(* LS Electric XG5000 project: PLC *)
(* PLC LSPLC *)

PROGRAM NewProgram (* task: 스캔 프로그램 *)
VAR
    Array_g : ARRAY[0..9] OF INT;
    Array_w : ARRAY[0..9] OF INT;
    FIFO_g : FIFO_INT;
    FIFO_w : FIFO_INT;
    grade AT %MW800 : INT;
    INST : TOF;
    INST1 : TOF;
    INST10 : TOF;
    INST11 : TOF;
    INST12 : TOF;
    INST13 : TOF;
    INST14 : TOF;
    INST15 : TOF;
    INST16 : TOF;
    INST17 : TOF;
    INST18 : TOF;
    INST19 : TOF;
    INST2 : TOF;
    INST20 : TOF;
    INST21 : TON;
    INST22 : TON;
    INST23 : TON;
    INST24 : TOF;
    INST25 : TON;
    INST26 : TON;
    INST27 : TON;
    INST28 : TON;
    INST29 : TON;
    INST3 : TOF;
    INST30 : TON;
    INST31 : TON;
    INST32 : TON;
    INST33 : TON;
    INST34 : TON;
    INST35 : TON;
    INST36 : TON;
    INST37 : TON;
    INST38 : TON;
    INST39 : TON;
    INST4 : TOF;
    INST40 : TON;
    INST41 : TON;
    INST42 : TON;
    INST43 : TON;
    INST44 : TON;
    INST45 : TON;
    INST46 : TON;
    INST47 : TON;
    INST48 : TON;
    INST49 : TON;
    INST5 : TOF;
    INST50 : TON;
    INST51 : TON;
    INST52 : TON;
    INST53 : TON;
    INST54 : TON;
    INST55 : TON;
    INST56 : TON;
    INST6 : TOF;
    INST7 : TOF;
    INST8 : TOF;
    INST9 : TOF;
    INT1_g : INT;
    INT1_w : INT;
    INT2_g : INT;
    INT2_w : INT;
    INT_w : INT;
    IN_ARY AT %MW0 : ARRAY[0..3] OF INT;
    R : BOOL;
    STOP AT %IX0.0.1 : BOOL;
    STR1 : STRING;
    STR2 : STRING;
    SYSTEM_ON AT %IX0.0.0 : BOOL;
    weight AT %MW700 : INT;
    고_1_signal : BOOL;
    고_1_적재 : TON;
    고_1_적재량 : CTU_INT;
    고_1_적재상황 AT %QW0.3.0 : INT;
    고_2_signal : BOOL;
    고_2_적재 : TON;
    고_2_적재량 : CTU_INT;
    고_2_적재상황 AT %QW0.3.1 : INT;
    고_3_signal : BOOL;
    고_3_적재량 : CTU_INT;
    고_3_적재상황 AT %QW0.3.2 : INT;
    등급난수생성 : TON;
    등급난수생성1 : TON;
    라인 AT %QX0.1.30 : BOOL;
    무게난수생성 : TON;
    무게난수생성1 : TON;
    바닥1 AT %MX13 : BOOL;
    바닥1_a AT %QW0.6.3 : INT;
    바닥1_작동 : TON;
    바닥2 AT %MX14 : BOOL;
    바닥2_a AT %QW0.7.0 : INT;
    바닥2_작동 : TON;
    바닥3 AT %MX15 : BOOL;
    바닥3_a AT %QW0.7.1 : INT;
    바닥3_작동 : TON;
    바닥4 AT %MX16 : BOOL;
    바닥4_a AT %QW0.7.2 : INT;
    바닥4_작동 : TON;
    바닥5 AT %MX17 : BOOL;
    바닥5_a AT %QW0.7.3 : INT;
    바닥5_작동 : TON;
    바닥6 AT %MX18 : BOOL;
    바닥6_a AT %QW0.8.0 : INT;
    바닥6_작동 : TON;
    바닥7 AT %MX19 : BOOL;
    바닥7_a AT %QW0.8.1 : INT;
    바닥7_작동 : TON;
    바닥8 AT %MX20 : BOOL;
    바닥8_a AT %QW0.8.2 : INT;
    바닥8_작동 : TON;
    바닥9 AT %MX21 : BOOL;
    바닥9_a AT %QW0.8.3 : INT;
    바닥9_작동 : TON;
    바닥_9_적재 : TON;
    분류로봇1 AT %MX500 : BOOL;
    분류로봇1_작동 : TOF;
    분류로봇2 AT %MX510 : BOOL;
    분류로봇2_작동 : TOF;
    분류로봇3 AT %MX520 : BOOL;
    분류로봇3_작동 : TOF;
    분류로봇4 AT %MX530 : BOOL;
    분류로봇4_작동 : TOF;
    분류로봇5 AT %MX540 : BOOL;
    분류로봇5_작동 : TOF;
    분류로봇6 AT %MX550 : BOOL;
    분류로봇6_작동 : TOF;
    삼_고_적재상황 AT %QW1.3.2 : INT;
    삼_저_적재상황 AT %QW1.3.0 : INT;
    삼_중_적재상황 AT %QW1.3.1 : INT;
    생산_signal : BOOL;
    생산_signal_a AT %QW0.4.0 : INT;
    소터1 AT %MX4 : BOOL;
    소터10 AT %MX12 : BOOL;
    소터10_a AT %QW0.6.2 : INT;
    소터10_작동 : TON;
    소터11_작동 : TON;
    소터12_작동 : TON;
    소터13_작동 : TON;
    소터14_작동 : TON;
    소터1_a AT %QW0.4.1 : INT;
    소터1_작동 : TON;
    소터2 AT %MW20 : INT;
    소터2_a AT %QW0.4.2 : INT;
    소터2_신호 AT %QW0.9.0 : INT;
    소터3 AT %MX5 : BOOL;
    소터3_a AT %QW0.4.3 : INT;
    소터3_작동 : TON;
    소터4 AT %MX6 : BOOL;
    소터4_a AT %QW0.5.0 : INT;
    소터4_작동 : TON;
    소터5 AT %MX7 : BOOL;
    소터5_a AT %QW0.5.1 : INT;
    소터5_작동 : TON;
    소터6 AT %MX8 : BOOL;
    소터6_a AT %QW0.5.2 : INT;
    소터6_작동 : TON;
    소터7 AT %MX9 : BOOL;
    소터7_a AT %QW0.5.3 : INT;
    소터7_작동 : TON;
    소터8 AT %MX10 : BOOL;
    소터8_a AT %QW0.6.0 : INT;
    소터8_작동 : TON;
    소터9 AT %MX11 : BOOL;
    소터9_a AT %QW0.6.1 : INT;
    소터9_작동 : TON;
    신호 AT %MX400 : BOOL;
    신호1 : BOOL;
    이_고_적재상황 AT %QW1.2.2 : INT;
    이_저_적재상황 AT %QW1.2.0 : INT;
    이_중_적재상황 AT %QW1.2.1 : INT;
    일_고_적재상황 AT %QW1.1.2 : INT;
    일_저_적재상황 AT %QW1.1.0 : INT;
    일_중_적재상황 AT %QW1.1.1 : INT;
    재생산_delay : TOF;
    재생산_signal AT %MX350 : BOOL;
    저_1_signal : BOOL;
    저_1_적재 : TON;
    저_1_적재량 : CTU_INT;
    저_1_적재상황 AT %QW0.1.0 : INT;
    저_2_signal : BOOL;
    저_2_적재 : TON;
    저_2_적재량 : CTU_INT;
    저_2_적재상황 AT %QW0.1.1 : INT;
    저_3_signal : BOOL;
    저_3_적재 : TON;
    저_3_적재량 : CTU_INT;
    저_3_적재상황 AT %QW0.1.2 : INT;
    저_4_적재량 : CTU_INT;
    저_5_적재량 : CTU_INT;
    저_6_적재량 : CTU_INT;
    저_7_적재량 : CTU_INT;
    저_8_적재량 : CTU_INT;
    저_9_적재 : TON;
    저_9_적재량 : CTU_INT;
    제품생산 : TP;
    중_1_signal : BOOL;
    중_1_적재 : TON;
    중_1_적재량 : CTU_INT;
    중_1_적재상황 AT %QW0.2.0 : INT;
    중_2_signal : BOOL;
    중_2_적재 : TON;
    중_2_적재량 : CTU_INT;
    중_2_적재상황 AT %QW0.2.1 : INT;
    중_3_signal : BOOL;
    중_3_적재량 : CTU_INT;
    중_3_적재상황 AT %QW0.2.2 : INT;
    품질로봇 AT %MW30 : INT;
    품질로봇가동 : TOF;
    품질로봇대기 : TON;
END_VAR
VAR
    _t1 : BOOL;
    _e2 : R_TRIG;
    _e3 : F_TRIG;
    _e4 : R_TRIG;
    _e5 : F_TRIG;
    _e6 : F_TRIG;
    _e7 : R_TRIG;
    _t8 : BOOL;
    _t9 : BOOL;
    _t10 : BOOL;
    _t11 : BOOL;
    _t12 : DINT;
    _t13 : BOOL;
    _t14 : BOOL;
    _t15 : BOOL;
    _t16 : BOOL;
    _t17 : BOOL;
    _t18 : DINT;
    _t19 : BOOL;
    _t20 : BOOL;
    _t21 : BOOL;
    _t22 : BOOL;
    _t23 : BOOL;
    _t24 : DINT;
    _t25 : BOOL;
    _t26 : BOOL;
    _t27 : BOOL;
    _t28 : BOOL;
    _t29 : BOOL;
    _t30 : BOOL;
    _t31 : BOOL;
    _t32 : BOOL;
    _t33 : BOOL;
    _t34 : BOOL;
    _t35 : BOOL;
    _t36 : BOOL;
    _e37 : R_TRIG;
    _e38 : R_TRIG;
    _e39 : R_TRIG;
    _e40 : R_TRIG;
    _e41 : R_TRIG;
    _e42 : R_TRIG;
    _e43 : R_TRIG;
    _e44 : R_TRIG;
    _e45 : R_TRIG;
    _t46 : BOOL;
END_VAR

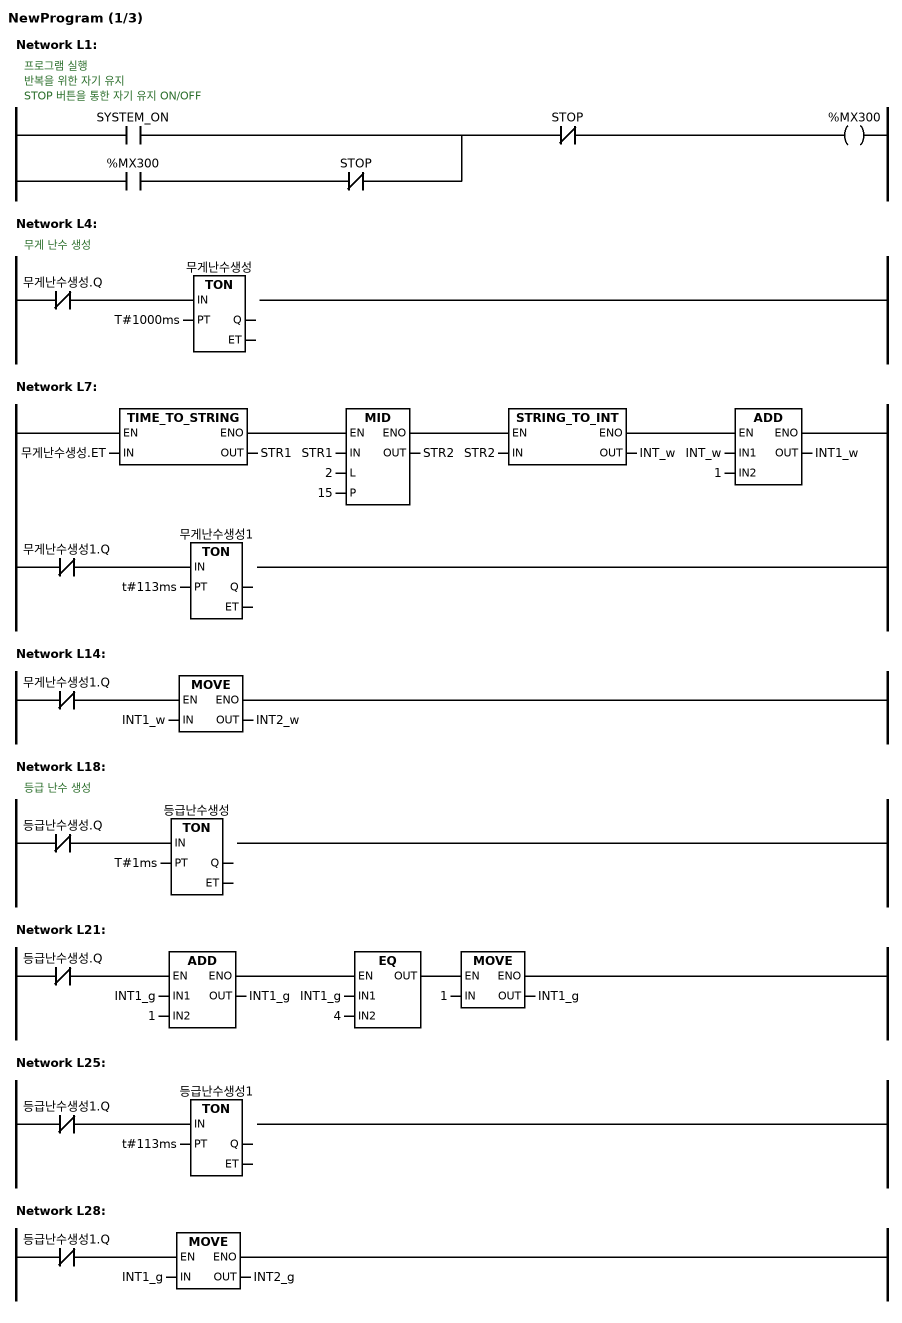
(* 프로그램 실행 / 반복을 위한 자기 유지 / STOP 버튼을 통한 자기 유지 ON/OFF *)
(* Rung L1 *)
%MX300 := (SYSTEM_ON OR (%MX300 AND NOT STOP)) AND NOT STOP;
(* 무게 난수 생성 *)
(* Rung L4 *)
무게난수생성(IN := NOT 무게난수생성.Q, PT := T#1000ms);
(* Rung L7 *)
STR1 := TIME_TO_STRING(무게난수생성.ET);
STR2 := MID(IN := STR1, L := 2, P := 15);
INT_w := STRING_TO_INT(STR2);
INT1_w := INT_w + 1;
무게난수생성1(IN := NOT 무게난수생성1.Q, PT := t#113ms);
(* Rung L14 *)
IF NOT 무게난수생성1.Q THEN INT2_w := INT1_w; END_IF;
(* 등급 난수 생성 *)
(* Rung L18 *)
등급난수생성(IN := NOT 등급난수생성.Q, PT := T#1ms);
(* Rung L21 *)
IF NOT 등급난수생성.Q THEN
    INT1_g := INT1_g + 1;
    _t1 := INT1_g = 4;
END_IF;
IF _t1 THEN INT1_g := 1; END_IF;
(* Rung L25 *)
등급난수생성1(IN := NOT 등급난수생성1.Q, PT := t#113ms);
(* Rung L28 *)
IF NOT 등급난수생성1.Q THEN INT2_g := INT1_g; END_IF;

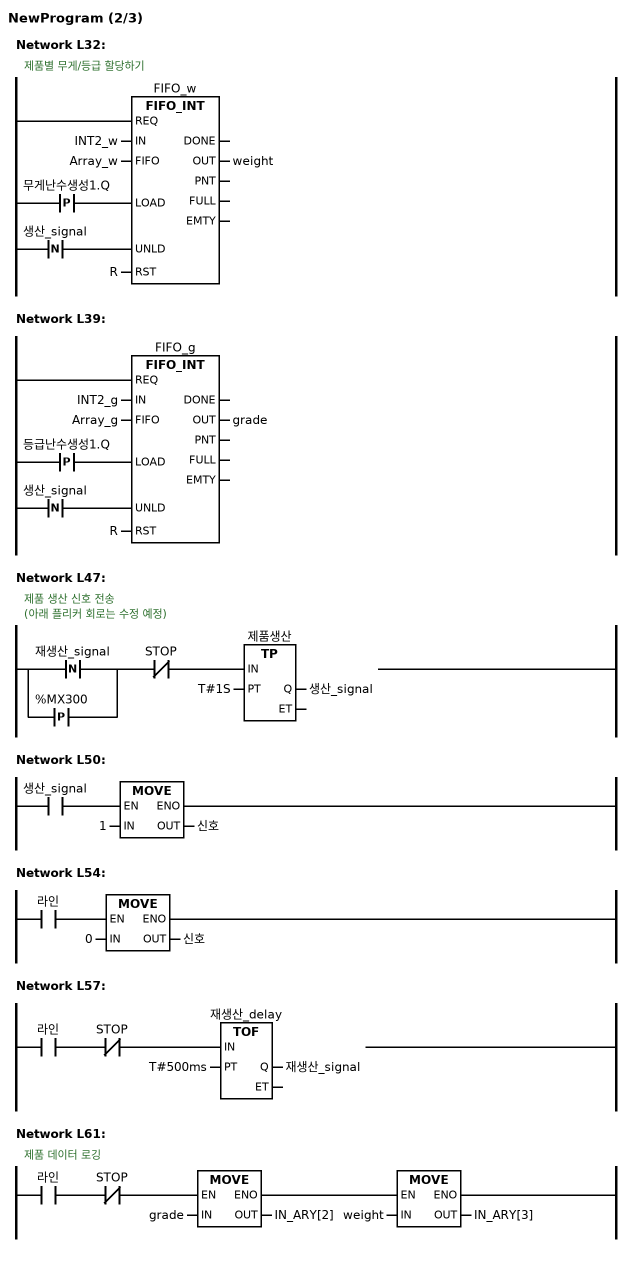
(* 제품별 무게/등급 할당하기 *)
(* Rung L32 *)
_e2(CLK := 무게난수생성1.Q);
_e3(CLK := 생산_signal);
FIFO_w(REQ := TRUE, IN := INT2_w, FIFO := Array_w, LOAD := _e2.Q, UNLD := _e3.Q, RST := R, OUT => weight);
(* Rung L39 *)
_e4(CLK := 등급난수생성1.Q);
_e5(CLK := 생산_signal);
FIFO_g(REQ := TRUE, IN := INT2_g, FIFO := Array_g, LOAD := _e4.Q, UNLD := _e5.Q, RST := R, OUT => grade);
(* 제품 생산 신호 전송 / (아래 플리커 회로는 수정 예정) *)
(* Rung L47 *)
_e6(CLK := 재생산_signal);
_e7(CLK := %MX300);
제품생산(IN := (_e6.Q OR _e7.Q) AND NOT STOP, PT := T#1S, Q => 생산_signal);
(* Rung L50 *)
IF 생산_signal THEN 신호 := 1; END_IF;
(* Rung L54 *)
IF 라인 THEN 신호 := 0; END_IF;
(* Rung L57 *)
재생산_delay(IN := 라인 AND NOT STOP, PT := T#500ms, Q => 재생산_signal);
(* 제품 데이터 로깅 *)
(* Rung L61 *)
IF 라인 AND NOT STOP THEN
    IN_ARY[2] := grade;
    IN_ARY[3] := weight;
END_IF;

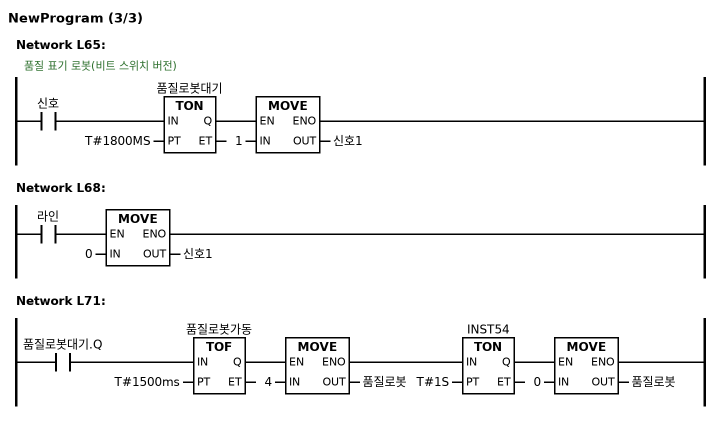
(* 품질 표기 로봇(비트 스위치 버전) *)
(* Rung L65 *)
품질로봇대기(IN := 신호, PT := T#1800MS);
IF 품질로봇대기.Q THEN 신호1 := 1; END_IF;
(* Rung L68 *)
IF 라인 THEN 신호1 := 0; END_IF;
(* Rung L71 *)
품질로봇가동(IN := 품질로봇대기.Q, PT := T#1500ms);
IF 품질로봇가동.Q THEN 품질로봇 := 4; END_IF;
INST54(IN := 품질로봇가동.Q, PT := T#1S);
IF INST54.Q THEN 품질로봇 := 0; END_IF;

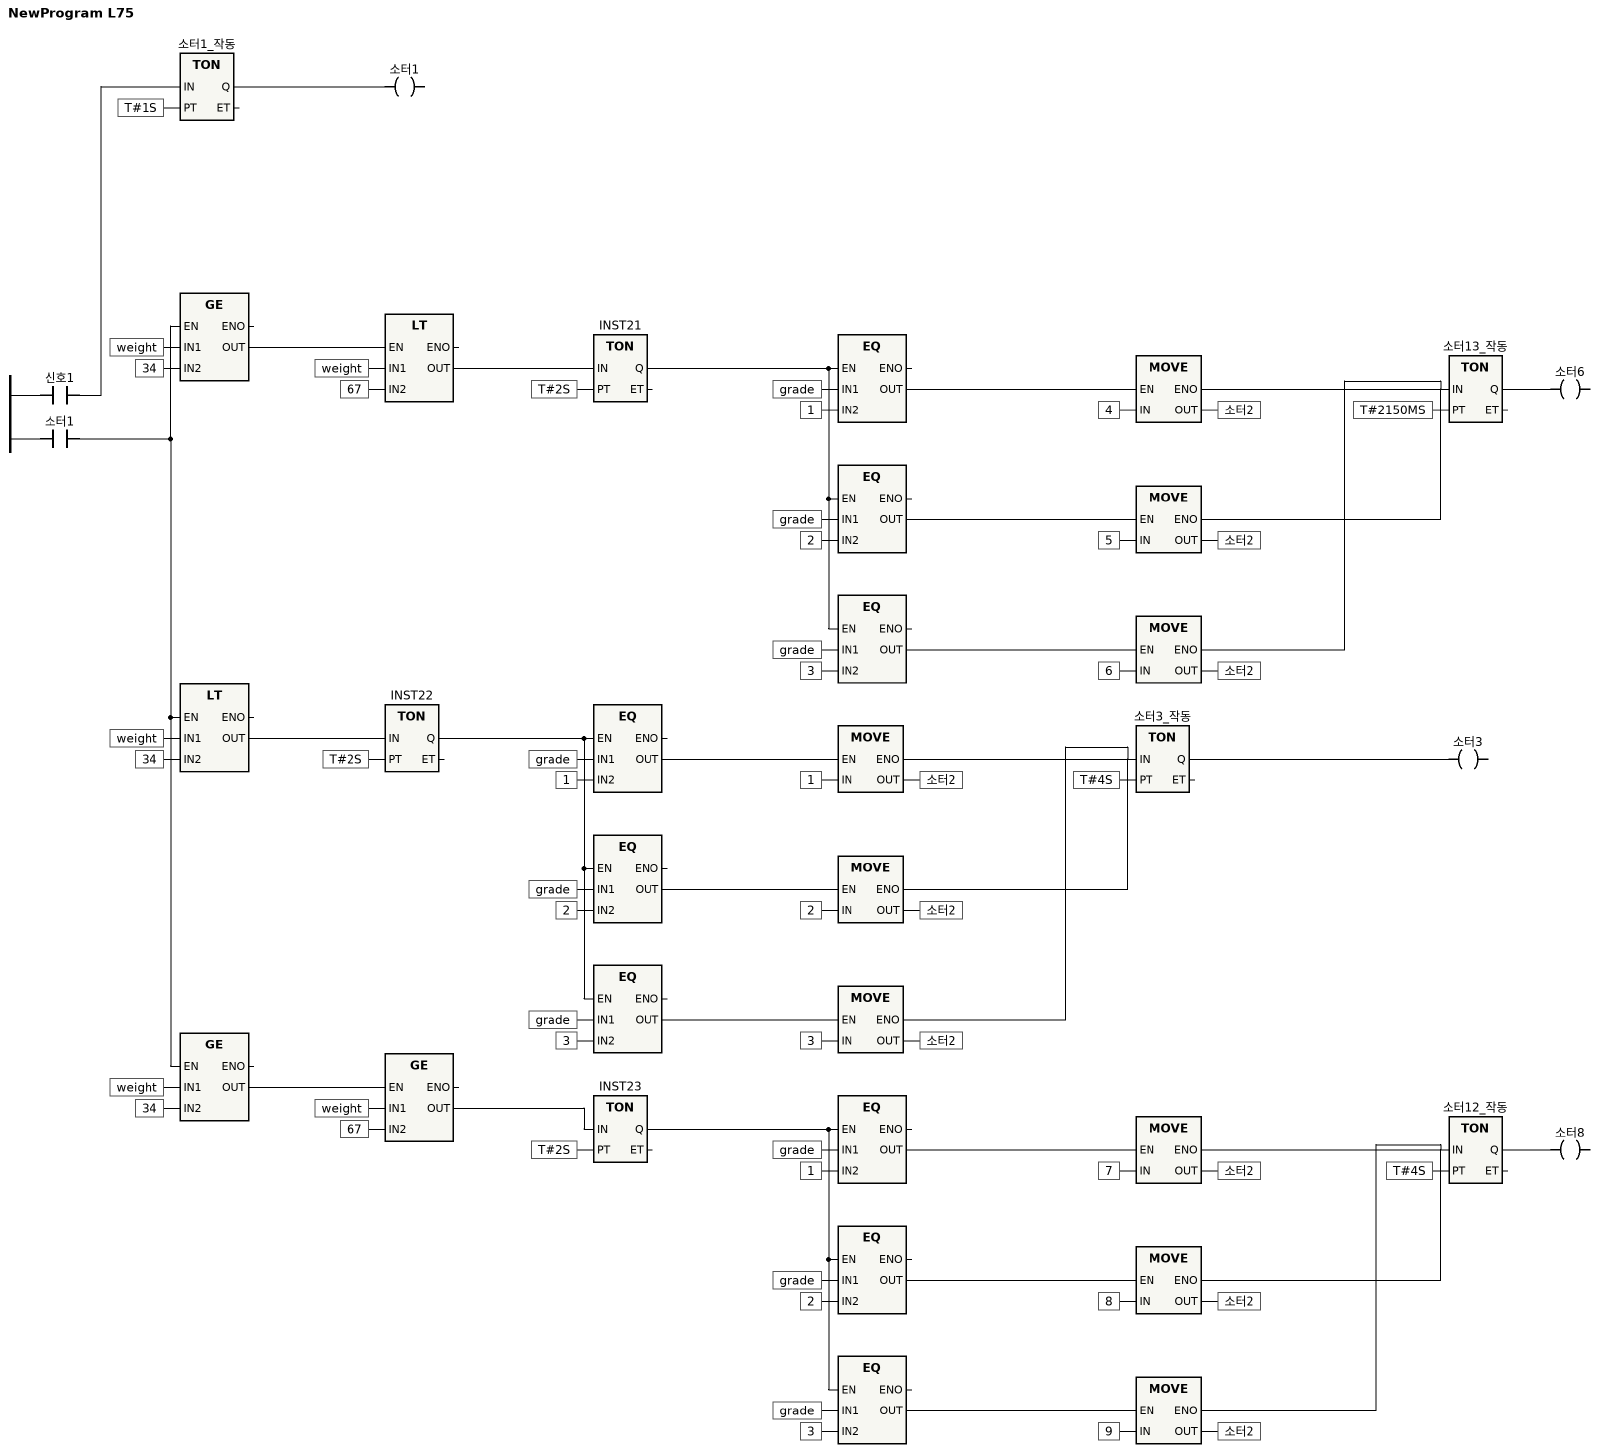
(* 등급/무게별 제품 분류 *)
(* Rung L75 *)
소터1_작동(IN := 신호1, PT := T#1S);
소터1 := 소터1_작동.Q;
IF 소터1 THEN _t8 := weight < 34; END_IF;
INST22(IN := _t8, PT := T#2S);
IF INST22.Q THEN _t9 := grade = 1; END_IF;
IF _t9 THEN 소터2 := 1; END_IF;
IF INST22.Q THEN _t10 := grade = 2; END_IF;
IF _t10 THEN 소터2 := 2; END_IF;
IF INST22.Q THEN _t11 := grade = 3; END_IF;
_t12 := 소터2;
IF _t11 THEN 소터2 := 3; END_IF;
소터3_작동(IN := _t9 OR _t10 OR _t11, PT := T#4S);
소터3 := 소터3_작동.Q;
IF 소터1 THEN _t13 := weight >= 34; END_IF;
IF _t13 THEN _t14 := weight < 67; END_IF;
INST21(IN := _t14, PT := T#2S);
IF INST21.Q THEN _t15 := grade = 1; END_IF;
IF _t15 THEN 소터2 := 4; END_IF;
IF INST21.Q THEN _t16 := grade = 2; END_IF;
IF _t16 THEN 소터2 := 5; END_IF;
IF INST21.Q THEN _t17 := grade = 3; END_IF;
_t18 := 소터2;
IF _t17 THEN 소터2 := 6; END_IF;
소터13_작동(IN := _t15 OR _t16 OR _t17, PT := T#2150MS);
소터6 := 소터13_작동.Q;
IF 소터1 THEN _t19 := weight >= 34; END_IF;
IF _t19 THEN _t20 := weight >= 67; END_IF;
INST23(IN := _t20, PT := T#2S);
IF INST23.Q THEN _t21 := grade = 1; END_IF;
IF _t21 THEN 소터2 := 7; END_IF;
IF INST23.Q THEN _t22 := grade = 2; END_IF;
IF _t22 THEN 소터2 := 8; END_IF;
IF INST23.Q THEN _t23 := grade = 3; END_IF;
_t24 := 소터2;
IF _t23 THEN 소터2 := 9; END_IF;
소터12_작동(IN := _t21 OR _t22 OR _t23, PT := T#4S);
소터8 := 소터12_작동.Q;

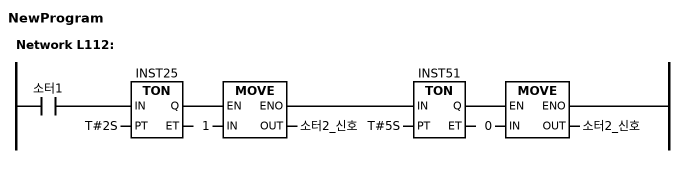
(* Rung L112 *)
INST25(IN := 소터1, PT := T#2S);
IF INST25.Q THEN 소터2_신호 := 1; END_IF;
INST51(IN := INST25.Q, PT := T#5S);
IF INST51.Q THEN 소터2_신호 := 0; END_IF;

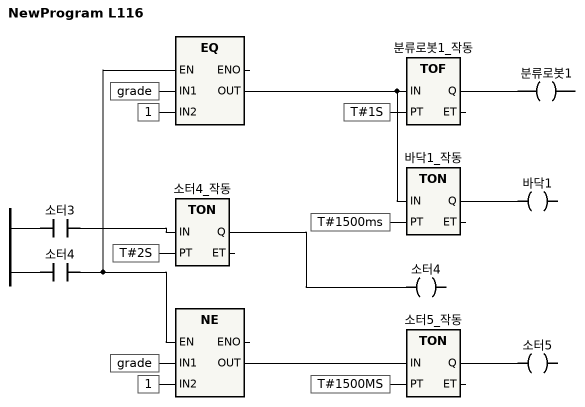
(* 저분류 *)
(* Rung L116 *)
소터4_작동(IN := 소터3, PT := T#2S);
소터4 := 소터4_작동.Q;
IF 소터4 THEN _t25 := grade = 1; END_IF;
분류로봇1_작동(IN := _t25, PT := T#1S);
분류로봇1 := 분류로봇1_작동.Q;
바닥1_작동(IN := _t25, PT := T#1500ms);
바닥1 := 바닥1_작동.Q;
IF 소터4 THEN _t26 := grade <> 1; END_IF;
소터5_작동(IN := _t26, PT := T#1500MS);
소터5 := 소터5_작동.Q;

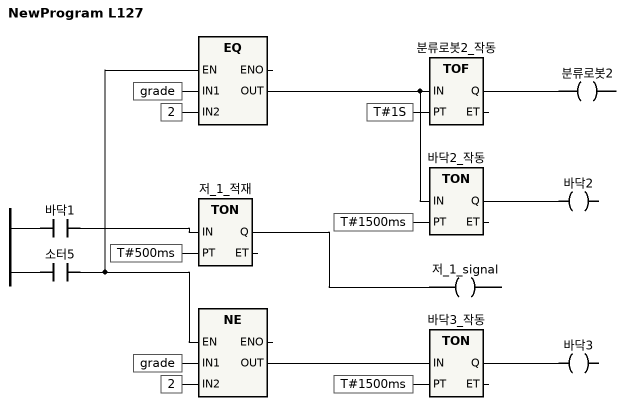
(* Rung L127 *)
저_1_적재(IN := 바닥1, PT := T#500ms);
저_1_signal := 저_1_적재.Q;
IF 소터5 THEN _t27 := grade = 2; END_IF;
분류로봇2_작동(IN := _t27, PT := T#1S);
분류로봇2 := 분류로봇2_작동.Q;
바닥2_작동(IN := _t27, PT := T#1500ms);
바닥2 := 바닥2_작동.Q;
IF 소터5 THEN _t28 := grade <> 2; END_IF;
바닥3_작동(IN := _t28, PT := T#1500ms);
바닥3 := 바닥3_작동.Q;

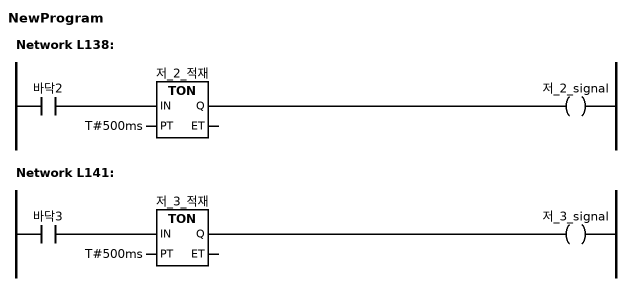
(* Rung L138 *)
저_2_적재(IN := 바닥2, PT := T#500ms);
저_2_signal := 저_2_적재.Q;
(* Rung L141 *)
저_3_적재(IN := 바닥3, PT := T#500ms);
저_3_signal := 저_3_적재.Q;

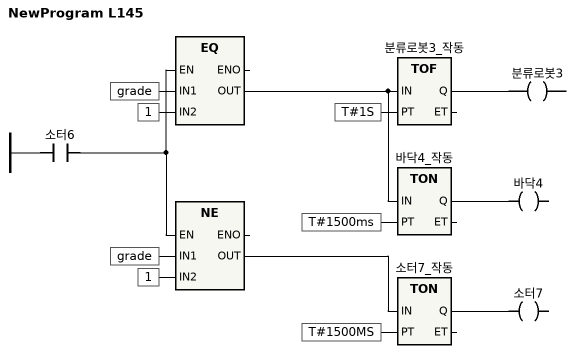
(* 중 분류 *)
(* Rung L145 *)
IF 소터6 THEN _t29 := grade = 1; END_IF;
분류로봇3_작동(IN := _t29, PT := T#1S);
분류로봇3 := 분류로봇3_작동.Q;
바닥4_작동(IN := _t29, PT := T#1500ms);
바닥4 := 바닥4_작동.Q;
IF 소터6 THEN _t30 := grade <> 1; END_IF;
소터7_작동(IN := _t30, PT := T#1500MS);
소터7 := 소터7_작동.Q;

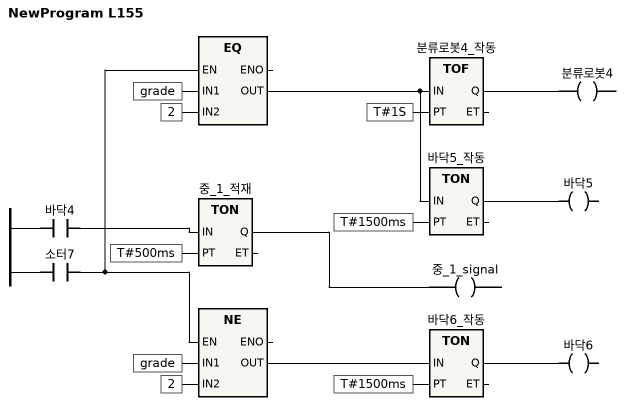
(* Rung L155 *)
중_1_적재(IN := 바닥4, PT := T#500ms);
중_1_signal := 중_1_적재.Q;
IF 소터7 THEN _t31 := grade = 2; END_IF;
분류로봇4_작동(IN := _t31, PT := T#1S);
분류로봇4 := 분류로봇4_작동.Q;
바닥5_작동(IN := _t31, PT := T#1500ms);
바닥5 := 바닥5_작동.Q;
IF 소터7 THEN _t32 := grade <> 2; END_IF;
바닥6_작동(IN := _t32, PT := T#1500ms);
바닥6 := 바닥6_작동.Q;

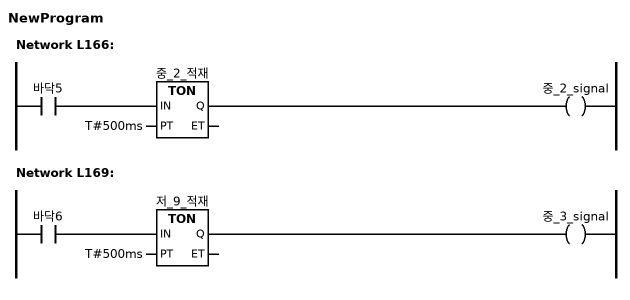
(* Rung L166 *)
중_2_적재(IN := 바닥5, PT := T#500ms);
중_2_signal := 중_2_적재.Q;
(* Rung L169 *)
저_9_적재(IN := 바닥6, PT := T#500ms);
중_3_signal := 저_9_적재.Q;

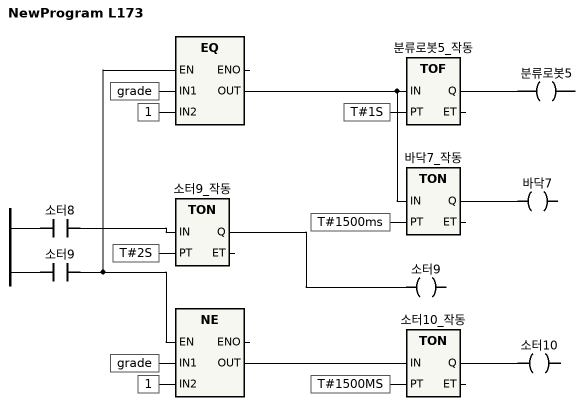
(* 고 분류 *)
(* Rung L173 *)
소터9_작동(IN := 소터8, PT := T#2S);
소터9 := 소터9_작동.Q;
IF 소터9 THEN _t33 := grade = 1; END_IF;
분류로봇5_작동(IN := _t33, PT := T#1S);
분류로봇5 := 분류로봇5_작동.Q;
바닥7_작동(IN := _t33, PT := T#1500ms);
바닥7 := 바닥7_작동.Q;
IF 소터9 THEN _t34 := grade <> 1; END_IF;
소터10_작동(IN := _t34, PT := T#1500MS);
소터10 := 소터10_작동.Q;

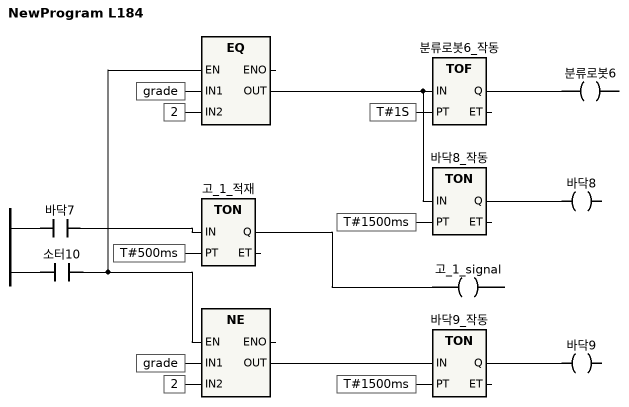
(* Rung L184 *)
고_1_적재(IN := 바닥7, PT := T#500ms);
고_1_signal := 고_1_적재.Q;
IF 소터10 THEN _t35 := grade = 2; END_IF;
분류로봇6_작동(IN := _t35, PT := T#1S);
분류로봇6 := 분류로봇6_작동.Q;
바닥8_작동(IN := _t35, PT := T#1500ms);
바닥8 := 바닥8_작동.Q;
IF 소터10 THEN _t36 := grade <> 2; END_IF;
바닥9_작동(IN := _t36, PT := T#1500ms);
바닥9 := 바닥9_작동.Q;

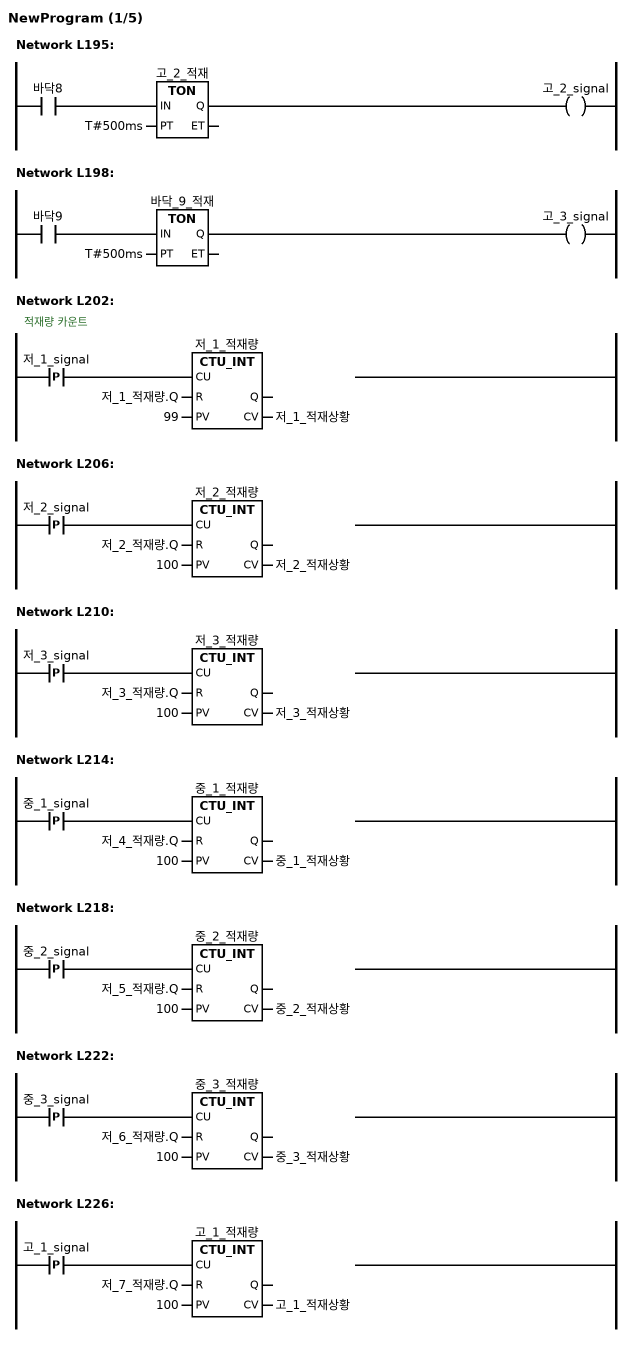
(* Rung L195 *)
고_2_적재(IN := 바닥8, PT := T#500ms);
고_2_signal := 고_2_적재.Q;
(* Rung L198 *)
바닥_9_적재(IN := 바닥9, PT := T#500ms);
고_3_signal := 바닥_9_적재.Q;
(* 적재량 카운트 *)
(* Rung L202 *)
_e37(CLK := 저_1_signal);
저_1_적재량(CU := _e37.Q, R := 저_1_적재량.Q, PV := 99, CV => 저_1_적재상황);
(* Rung L206 *)
_e38(CLK := 저_2_signal);
저_2_적재량(CU := _e38.Q, R := 저_2_적재량.Q, PV := 100, CV => 저_2_적재상황);
(* Rung L210 *)
_e39(CLK := 저_3_signal);
저_3_적재량(CU := _e39.Q, R := 저_3_적재량.Q, PV := 100, CV => 저_3_적재상황);
(* Rung L214 *)
_e40(CLK := 중_1_signal);
중_1_적재량(CU := _e40.Q, R := 저_4_적재량.Q, PV := 100, CV => 중_1_적재상황);
(* Rung L218 *)
_e41(CLK := 중_2_signal);
중_2_적재량(CU := _e41.Q, R := 저_5_적재량.Q, PV := 100, CV => 중_2_적재상황);
(* Rung L222 *)
_e42(CLK := 중_3_signal);
중_3_적재량(CU := _e42.Q, R := 저_6_적재량.Q, PV := 100, CV => 중_3_적재상황);
(* Rung L226 *)
_e43(CLK := 고_1_signal);
고_1_적재량(CU := _e43.Q, R := 저_7_적재량.Q, PV := 100, CV => 고_1_적재상황);

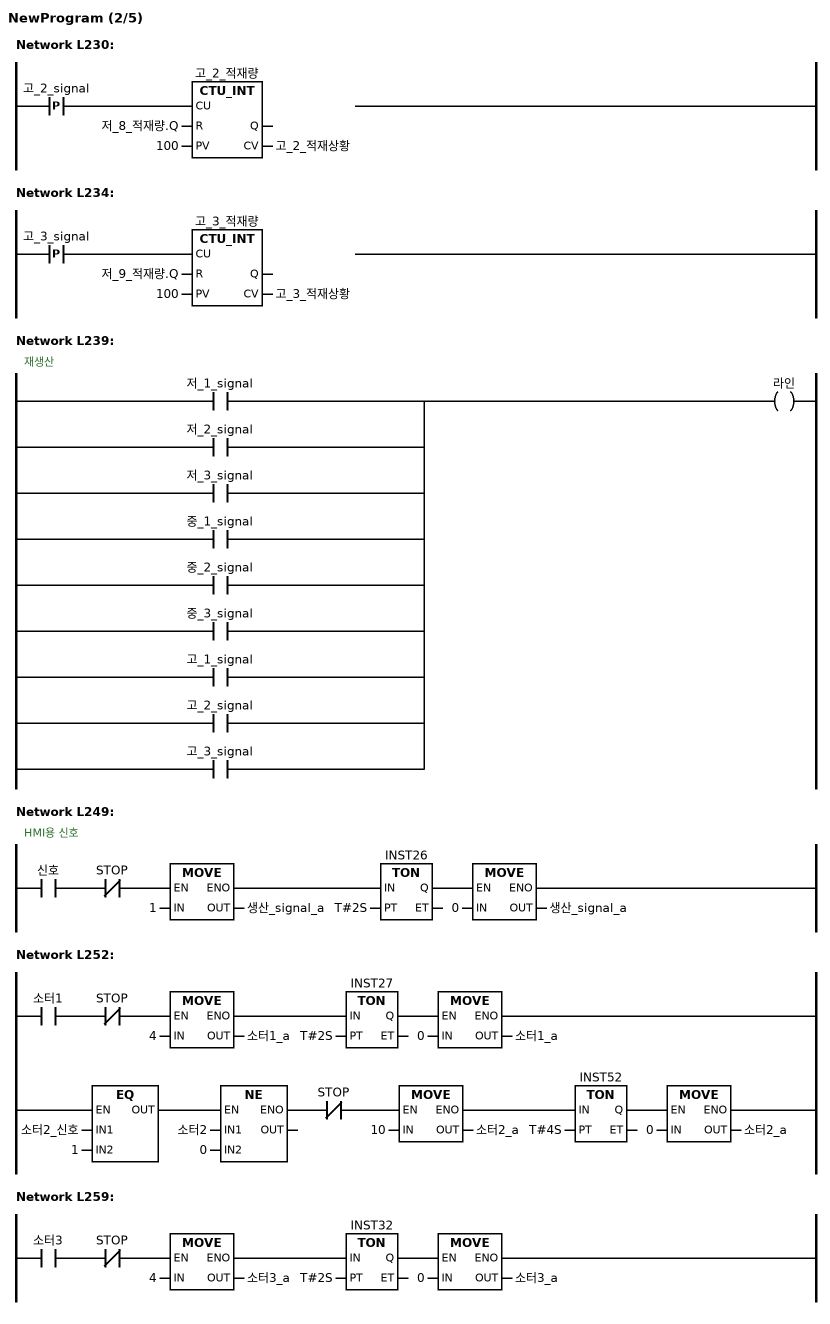
(* Rung L230 *)
_e44(CLK := 고_2_signal);
고_2_적재량(CU := _e44.Q, R := 저_8_적재량.Q, PV := 100, CV => 고_2_적재상황);
(* Rung L234 *)
_e45(CLK := 고_3_signal);
고_3_적재량(CU := _e45.Q, R := 저_9_적재량.Q, PV := 100, CV => 고_3_적재상황);
(* 재생산 *)
(* Rung L239 *)
라인 := 저_1_signal OR 저_2_signal OR 저_3_signal OR 중_1_signal OR 중_2_signal OR 중_3_signal OR 고_1_signal OR 고_2_signal OR 고_3_signal;
(* HMI용 신호 *)
(* Rung L249 *)
IF 신호 AND NOT STOP THEN 생산_signal_a := 1; END_IF;
INST26(IN := 신호 AND NOT STOP, PT := T#2S);
IF INST26.Q THEN 생산_signal_a := 0; END_IF;
(* Rung L252 *)
IF 소터1 AND NOT STOP THEN 소터1_a := 4; END_IF;
INST27(IN := 소터1 AND NOT STOP, PT := T#2S);
IF INST27.Q THEN 소터1_a := 0; END_IF;
IF 소터2_신호 = 1 THEN _t46 := 소터2 <> 0; END_IF;
IF (소터2_신호 = 1) AND NOT STOP THEN 소터2_a := 10; END_IF;
INST52(IN := (소터2_신호 = 1) AND NOT STOP, PT := T#4S);
IF INST52.Q THEN 소터2_a := 0; END_IF;
(* Rung L259 *)
IF 소터3 AND NOT STOP THEN 소터3_a := 4; END_IF;
INST32(IN := 소터3 AND NOT STOP, PT := T#2S);
IF INST32.Q THEN 소터3_a := 0; END_IF;

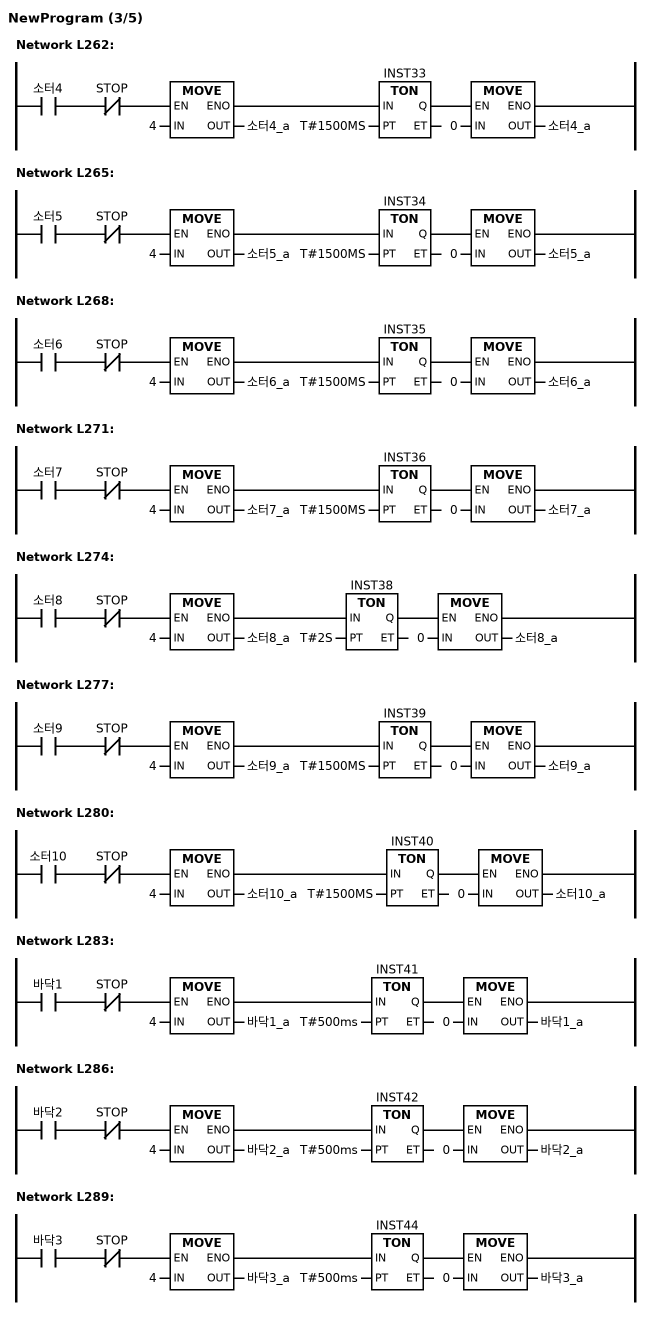
(* Rung L262 *)
IF 소터4 AND NOT STOP THEN 소터4_a := 4; END_IF;
INST33(IN := 소터4 AND NOT STOP, PT := T#1500MS);
IF INST33.Q THEN 소터4_a := 0; END_IF;
(* Rung L265 *)
IF 소터5 AND NOT STOP THEN 소터5_a := 4; END_IF;
INST34(IN := 소터5 AND NOT STOP, PT := T#1500MS);
IF INST34.Q THEN 소터5_a := 0; END_IF;
(* Rung L268 *)
IF 소터6 AND NOT STOP THEN 소터6_a := 4; END_IF;
INST35(IN := 소터6 AND NOT STOP, PT := T#1500MS);
IF INST35.Q THEN 소터6_a := 0; END_IF;
(* Rung L271 *)
IF 소터7 AND NOT STOP THEN 소터7_a := 4; END_IF;
INST36(IN := 소터7 AND NOT STOP, PT := T#1500MS);
IF INST36.Q THEN 소터7_a := 0; END_IF;
(* Rung L274 *)
IF 소터8 AND NOT STOP THEN 소터8_a := 4; END_IF;
INST38(IN := 소터8 AND NOT STOP, PT := T#2S);
IF INST38.Q THEN 소터8_a := 0; END_IF;
(* Rung L277 *)
IF 소터9 AND NOT STOP THEN 소터9_a := 4; END_IF;
INST39(IN := 소터9 AND NOT STOP, PT := T#1500MS);
IF INST39.Q THEN 소터9_a := 0; END_IF;
(* Rung L280 *)
IF 소터10 AND NOT STOP THEN 소터10_a := 4; END_IF;
INST40(IN := 소터10 AND NOT STOP, PT := T#1500MS);
IF INST40.Q THEN 소터10_a := 0; END_IF;
(* Rung L283 *)
IF 바닥1 AND NOT STOP THEN 바닥1_a := 4; END_IF;
INST41(IN := 바닥1 AND NOT STOP, PT := T#500ms);
IF INST41.Q THEN 바닥1_a := 0; END_IF;
(* Rung L286 *)
IF 바닥2 AND NOT STOP THEN 바닥2_a := 4; END_IF;
INST42(IN := 바닥2 AND NOT STOP, PT := T#500ms);
IF INST42.Q THEN 바닥2_a := 0; END_IF;
(* Rung L289 *)
IF 바닥3 AND NOT STOP THEN 바닥3_a := 4; END_IF;
INST44(IN := 바닥3 AND NOT STOP, PT := T#500ms);
IF INST44.Q THEN 바닥3_a := 0; END_IF;

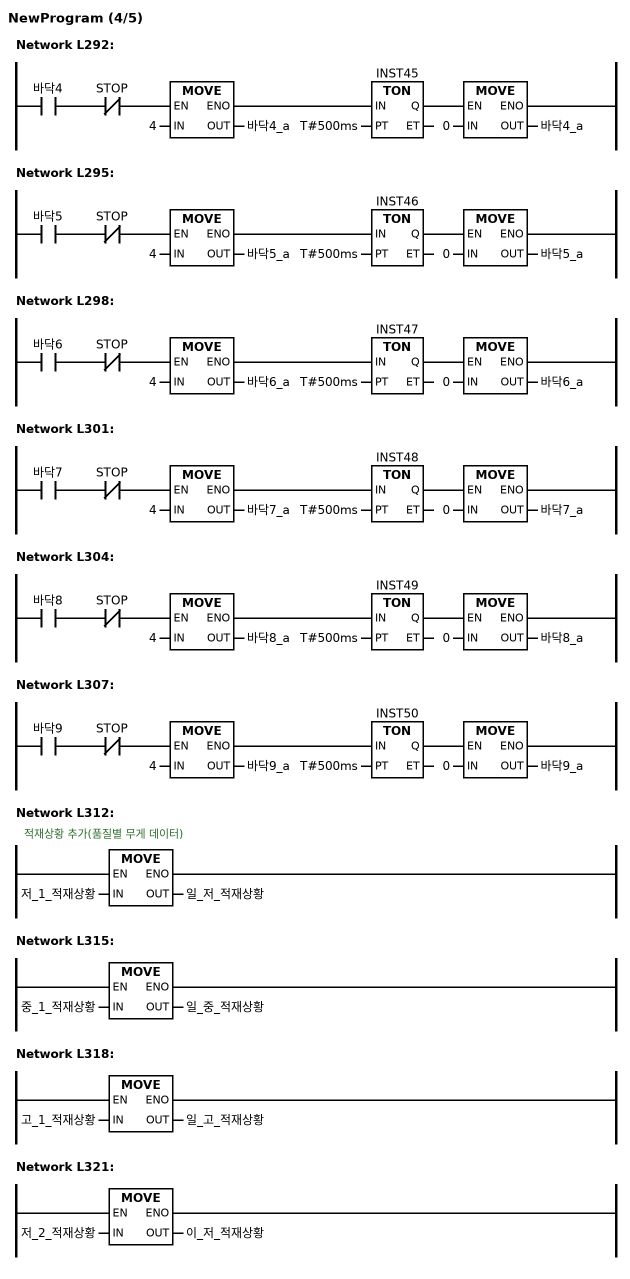
(* Rung L292 *)
IF 바닥4 AND NOT STOP THEN 바닥4_a := 4; END_IF;
INST45(IN := 바닥4 AND NOT STOP, PT := T#500ms);
IF INST45.Q THEN 바닥4_a := 0; END_IF;
(* Rung L295 *)
IF 바닥5 AND NOT STOP THEN 바닥5_a := 4; END_IF;
INST46(IN := 바닥5 AND NOT STOP, PT := T#500ms);
IF INST46.Q THEN 바닥5_a := 0; END_IF;
(* Rung L298 *)
IF 바닥6 AND NOT STOP THEN 바닥6_a := 4; END_IF;
INST47(IN := 바닥6 AND NOT STOP, PT := T#500ms);
IF INST47.Q THEN 바닥6_a := 0; END_IF;
(* Rung L301 *)
IF 바닥7 AND NOT STOP THEN 바닥7_a := 4; END_IF;
INST48(IN := 바닥7 AND NOT STOP, PT := T#500ms);
IF INST48.Q THEN 바닥7_a := 0; END_IF;
(* Rung L304 *)
IF 바닥8 AND NOT STOP THEN 바닥8_a := 4; END_IF;
INST49(IN := 바닥8 AND NOT STOP, PT := T#500ms);
IF INST49.Q THEN 바닥8_a := 0; END_IF;
(* Rung L307 *)
IF 바닥9 AND NOT STOP THEN 바닥9_a := 4; END_IF;
INST50(IN := 바닥9 AND NOT STOP, PT := T#500ms);
IF INST50.Q THEN 바닥9_a := 0; END_IF;
(* 적재상황 추가(품질별 무게 데이터) *)
(* Rung L312 *)
일_저_적재상황 := 저_1_적재상황;
(* Rung L315 *)
일_중_적재상황 := 중_1_적재상황;
(* Rung L318 *)
일_고_적재상황 := 고_1_적재상황;
(* Rung L321 *)
이_저_적재상황 := 저_2_적재상황;

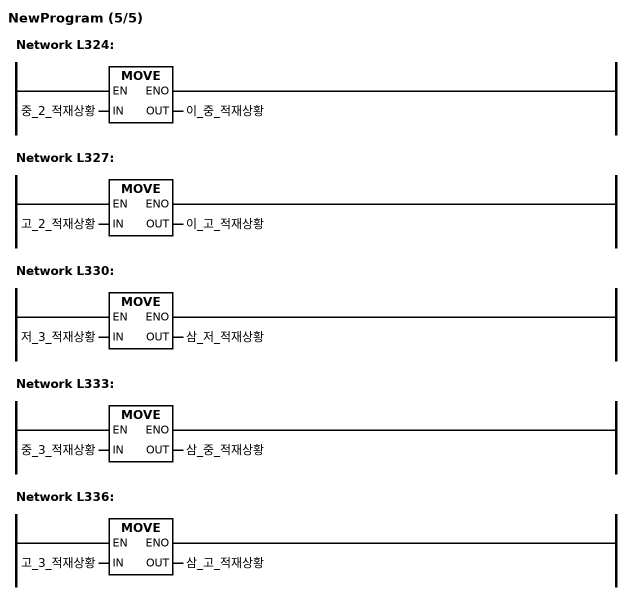
(* Rung L324 *)
이_중_적재상황 := 중_2_적재상황;
(* Rung L327 *)
이_고_적재상황 := 고_2_적재상황;
(* Rung L330 *)
삼_저_적재상황 := 저_3_적재상황;
(* Rung L333 *)
삼_중_적재상황 := 중_3_적재상황;
(* Rung L336 *)
삼_고_적재상황 := 고_3_적재상황;
END_PROGRAM